INTERFACE itfAxisCommand EXTENDS itfCommand

METHOD Update : MC_Error
VAR_INPUT
	Position: REAL;
	Velocity: REAL;
	EndVelocity: REAL;
	Acceleration: REAL;
	Deceleration: REAL;
	Jerk: REAL;
END_VAR
END_METHOD

END_INTERFACE

(* stored: Version 1.1.0.1, ProductVersion 3.1.4024.12
   Itf itfAxisCommand: Id {bfca13e7-409d-4156-8fc6-fcd16d016e02}
   Method Update: Id {22743afd-e290-4db2-9fd2-008534041ac5} *)
